// TIA Portal V17 export
// export: Created 2022-09-30T08:29:44.2144833Z, ExportSetting WithDefaults, DisplayName Totally Integrated Automation Portal, DisplayVersion V17 Update 5, DisplayName TIA Portal Openness, DisplayVersion V17 Update 5, DisplayName TIA Portal Teamcenter Gateway, DisplayVersion V17 Update 5, DisplayName TIA Portal Version Control Interface, DisplayVersion V17, DisplayName TIA Portal Test Suite Advanced, DisplayVersion V17 Update 1, DisplayName SINAMICS Startdrive Advanced, DisplayVersion V17 Update2, DisplayName SINAMICS Startdrive G130, G150, S120, S150, SINAMICS MV, S210, DisplayVersion V17 Update2, DisplayName SINAMICS Startdrive G110M, G120, G120C, G120D, G120P, G115D, DisplayVersion V17 Update2, DisplayName STEP 7 Professional, DisplayVersion V17 Update 5, DisplayName STEP 7 CFC, DisplayVersion V17 Update 1, DisplayName STEP 7 Safety, DisplayVersion V17, DisplayName WinCC Advanced / Unified PC, DisplayVersion V17 Update 5, DisplayName WinCC Unified Calendar, DisplayVersion V17, DisplayName WinCC Unified Performance Insight, DisplayVersion V17
FUNCTION "FC_CALCUL" : Void   // FC1, LAD
{ S7_Optimized_Access := 'TRUE' }
VERSION : 0.1
// FC Calcul
// stored: AutoNumber true, IsIECCheckEnabled false, SetENOAutomatically false, UDAEnableTagReadback false
   VAR_INPUT
      Validation : Bool;
   END_VAR
   VAR_IN_OUT
      DATA : "UDT_CALCUL";
   END_VAR
   VAR CONSTANT
      PI : Real := 3.1416;
   END_VAR
BEGIN

REGION Network 1: Calcul de base
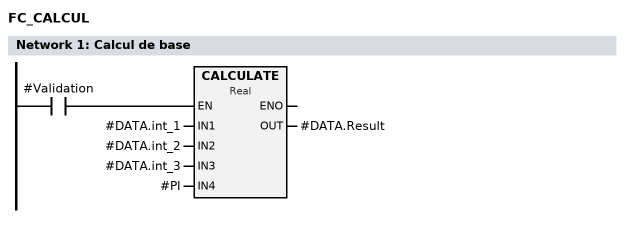
   RUNG wire#powerrail
      Contact( #Validation )
      { S7_Templates := "SrcType := Real"; S7_Expression := "((IN1 / IN2)+IN3)*IN4" } Calculate(in1 := #DATA.int_1, in2 := #DATA.int_2, in3 := #DATA.int_3, in4 := #PI, out => #DATA.Result)
   END_RUNG
   // the same network as SCL:
   IF #Validation THEN #DATA.Result := ((#DATA.int_1 / #DATA.int_2)+#DATA.int_3)*#PI; END_IF;
END_REGION

REGION Network 2 (SCL): Erreur DIV/0
   IF (#DATA.int_2 =0) AND #Validation  THEN  //SI dividende = 0
       #DATA.Result := (INT_TO_REAL(#DATA.int_1)  + #DATA.Real) * #PI;
       ;
   END_IF;
END_REGION
END_FUNCTION
